// TIA Portal V20 export
// export: Created 2025-12-01T14:57:13.3377999Z, ExportSetting None, DisplayName Totally Integrated Automation Portal, DisplayVersion V20 Update 3, DisplayName TIA Portal Openness, DisplayVersion V20 Update 3, DisplayName TIA Portal Version Control Interface, DisplayVersion V20 Update 3, DisplayName STEP 7 Professional, DisplayVersion V20 Update 3, DisplayName STEP 7 Safety, DisplayVersion V20 Update 2, DisplayName WinCC Basic/Comfort/Advanced, DisplayVersion V20 Update 3, DisplayName WinCC Professional, DisplayVersion V20 Update 3, DisplayName WinCC Unified, DisplayVersion V20 Update 3
FUNCTION "FC883_CalcularError_Armarios" : Void   // FC883, LAD
{ S7_Optimized_Access := 'FALSE' }
AUTHOR : ERRORES
NAME : 20160407
VERSION : 3.1
// stored: AutoNumber false, SetENOAutomatically false
   VAR_INPUT
      NumDB_Errores : UInt;
      Numero : UInt;
   END_VAR
   VAR_IN_OUT
      Codigo : UDInt;
      Emergencia : Bool;
      ErrorGrave : Bool;
      ErrorLeve : Bool;
   END_VAR
   VAR_TEMP
      ErrorFIFO : UDInt;
      P_Inicial : DWord;
      P_Final : DWord;
      NumDB : Word;
      Armario : UDInt;
      NumEmerg : UDInt;
      NumErrorGrave : UDInt;
      NumErrorLeve : UDInt;
      OffsetEmerg : UInt;
      OffsetErrorGrave : UInt;
      OffsetErrorLeve : UInt;
      MaxBitsGraves : UInt;
      MaxBitsLeves : UInt;
      LongBits : UInt;
      Zona : UInt;
   END_VAR
BEGIN

NETWORK
TITLE = Inicializar
///////////////////////////////////////////////////////////////////////////
// --- Inicializar Variables

      L     #NumDB_Errores;  // DB de Errores FIFO
      T     #NumDB;

      L     0;
      T     #NumEmerg;  // nieves 28/08/25      // No hay Emergencia (Inicial)
      T     #NumErrorLeve;  // No hay Error (Inicial)
      T     #NumErrorGrave;


      L     16;  // Long de la Estructura
      T     #LongBits;

      L     0;  // Offset de Los Bits
      T     #OffsetEmerg;
      L     2;
      T     #OffsetErrorGrave;
      L     4;
      T     #OffsetErrorLeve;

      L     15;  // Numero de Bits
      T     #MaxBitsGraves;
      L     95;
      T     #MaxBitsLeves;

      L     #Numero;
      T     #Zona;


///////////////////////////////////////////////////////////////////////////
// --- Comprobación del Numero de Dispositivo

      L     #Zona;
      L     0;
      <I;
      JC    Final;
      L     #Zona;
      L     "CTE_MaxDispositivos";
      >I;
      JC    Final;


///////////////////////////////////////////////////////////////////////////
// --- Calcular el Numero de Armario

      L     "CTE_OffsetCCPIF";
      L     100;
      *D;
      L     #Zona;
      +D;
      T     #Armario;

      JU    Mirar_EmergenciaGrave;  // Mirar a Emergencias Graves



NETWORK
TITLE = Codigo de Emegencia
Mirar_EmergenciaGrave:NOP   0;

///////////////////////////////////////////////////////////////////////////
// --- Preparar Puntero Inicial y Final

      L     #Zona;
      L     #LongBits;
      *D;
      L     #OffsetEmerg;
      +D;
      SLD   3;
      T     #P_Inicial;
      T     #P_Final;


///////////////////////////////////////////////////////////////////////////
// --- Recorrer el Arrray de Errores

Bucle_EmergenciaGrave:NOP   0;
      OPN   DB [#NumDB];  // Recorrer todos los Bits

      A     DBX [#P_Final];
      JC    Existe_EmergenciaGrave;  // Esta Activado este Bit

      L     #P_Final;
      L     #P_Inicial;
      -D;
      L     #MaxBitsGraves;
      ==I;
      JC    Final_EmergenciaGrave;  // Si ha recorrido todos los bits

      L     #P_Final;
      L     P#0.1;
      +D;
      T     #P_Final;
      JU    Bucle_EmergenciaGrave;  // Siguiente Bit


///////////////////////////////////////////////////////////////////////////
// --- Calcular el codigo

Existe_EmergenciaGrave:NOP   0;
      L     #P_Final;
      L     #P_Inicial;
      -D;
      L     1;  // Empieza 1 -> 16
      +D;
      T     #NumEmerg;  // Numero Bit Actrivado

      L     #NumEmerg;
      T     #ErrorFIFO;  // Codigo Final HMI


///////////////////////////////////////////////////////////////////////////
// ---      Escribir el Error
// ---      Preparar para Visualizar

      SET;
      S     #Emergencia;  // Activar Emergencia Grave

      L     #NumEmerg;  // Escribir Codigo
      T     #Codigo;

      L     #ErrorFIFO;
      T     "DB861_FIFO_Errores".ArmariosGraves[#Zona];

      JU    Final_EmergenciaGrave;  // Final


///////////////////////////////////////////////////////////////////////////
// --- No Hay EMergencia Grave

Final_EmergenciaGrave:NOP   0;  // No hay Graves
      JU    Mirar_ErrorGrave;  // Ir a Mirar los errores graves



NETWORK
TITLE = Codigo de Error de Grave
Mirar_ErrorGrave:NOP   0;

///////////////////////////////////////////////////////////////////////////
// --- Preparar Puntero Inicial y Final

      L     #Zona;
      L     #LongBits;
      *D;
      L     #OffsetErrorGrave;
      +D;
      SLD   3;
      T     #P_Inicial;
      T     #P_Final;


///////////////////////////////////////////////////////////////////////////
// --- Recorrer el Arrray de Errores

Bucle_ErrorGrave:NOP   0;
      OPN   DB [#NumDB];  // Recorrer todos los Bits
      A     DBX [#P_Final];
      JC    Existe_ErrorGrave;  // Esta Activado este Bit

      L     #P_Final;
      L     #P_Inicial;
      -D;
      L     #MaxBitsGraves;
      ==I;
      JC    Final_ErrorGrave;  // Si ha recorrido todos los bits

      L     #P_Final;
      L     P#0.1;
      +D;
      T     #P_Final;
      JU    Bucle_ErrorGrave;  // Siguiente Bit


///////////////////////////////////////////////////////////////////////////
// --- Calcular el Numero de Error

Existe_ErrorGrave:NOP   0;
      L     #P_Final;
      L     #P_Inicial;
      -D;
      L     100;  // Empieza 100 -> 199
      +D;
      T     #NumErrorGrave;  // Numero Bit Activado

      L     #NumErrorGrave;
      T     #ErrorFIFO;  // Codigo Final HMI

///////////////////////////////////////////////////////////////////////////
// ---      Escribir el Error
// ---      Preparar para Visualizar

      SET;
      S     #ErrorGrave;  // Activar Error Grave

      SET;
      A     #Emergencia;  // Escribir Codigo ?
      JC    NoActivarCodigo_ErrorGrave;

      L     #NumErrorGrave;
      T     #Codigo;

NoActivarCodigo_ErrorGrave:NOP   0;
      SET;
      A     #Emergencia;  // Guardar FIFO GRAVE ?
      JC    Final_ErrorGrave;

      L     #ErrorFIFO;
      T     "DB861_FIFO_Errores".ArmariosGraves[#Zona];

      JU    Final_ErrorGrave;  // Mirar Leves


///////////////////////////////////////////////////////////////////////////
// --- No Hay Error

Final_ErrorGrave:NOP   0;  // No hay Graves
      JU    MirarErrorLeve;  // Ir a Mirar los Leves



NETWORK
TITLE = Codigo de Error de Leves
///////////////////////////////////////////////////////////////////////////
// --- Preparar Puntero Inicial y Final

MirarErrorLeve:L     #Zona;
      L     #LongBits;
      *D;
      L     #OffsetErrorLeve;
      +D;
      SLD   3;
      T     #P_Inicial;
      T     #P_Final;  //nieves 28/08/25


///////////////////////////////////////////////////////////////////////////
// --- Recorrer el Arrray de Errores

Bucle_ErrorLeve:NOP   0;
      OPN   DB [#NumDB];  // Recorrer todos los Errores
      A     DBX [#P_Final];
      JC    Existe_ErrorLeve;  // Esta Activado este Bit

      L     #P_Final;
      L     #P_Inicial;
      -D;
      L     #MaxBitsLeves;
      ==I;
      JC    Final_ErrorLeve;  // Si ha recorrido todos los bits

      L     #P_Final;
      L     P#0.1;
      +D;
      T     #P_Final;
      JU    Bucle_ErrorLeve;  // Siguiente Bit


///////////////////////////////////////////////////////////////////////////
// --- Calcular el Numero de Error

Existe_ErrorLeve:NOP   0;
      L     #P_Final;
      L     #P_Inicial;
      -D;
      L     200;  //200 --> 299
      +D;
      T     #NumErrorLeve;  // Numero Bit Actrivado

      L     #NumErrorLeve;
      T     #ErrorFIFO;  // Codigo Final HMI


///////////////////////////////////////////////////////////////////////////
// ---      Escribir el Error
// ---      Preparar para Visualizar

      SET;
      S     #ErrorLeve;  // Activar Error Leve

      SET;
      A     #Emergencia;  // Escribir Codigo ?
      O     #ErrorGrave;
      JC    NoActivarCodigo_ErrorLeve;

      L     #NumErrorLeve;
      T     #Codigo;

NoActivarCodigo_ErrorLeve:NOP   0;
//      U     #Emergencia         // nieves comentado para que se activen tambien los errores leves aunque haya emergencia
//      SPB   Final

      L     #ErrorFIFO;
      T     "DB861_FIFO_Errores".ArmariosLeves[#Zona];

      JU    Final;  // No mirar más


///////////////////////////////////////////////////////////////////////////
// --- No Hay Error

Final_ErrorLeve:NOP   0;  // No hay Leves


///////////////////////////////////////////////////////////////////////////
// --- AUTO-REARME

      SET;
      R     #ErrorLeve;  // DesActivar Error Leve

      L     0;
      T     "DB861_FIFO_Errores".ArmariosLeves[#Zona];

      SET;
      A     #Emergencia;  // Borrado del Codigo ?
      O     #ErrorGrave;
      JC    Final;

      L     0;
      T     #Codigo;

      JU    Final;  // No hay mirar nadie más



NETWORK
TITLE = Finalizar
///////////////////////////////////////////////////////////////////////////
// --- Se acabo la Funcion

Final:NOP   0;



END_FUNCTION
